TYPE sCmd :
STRUCT
	boStop : BOOL;
	boReset :BOOL;
	boJobReset: BOOL;
	boRFIDComplete: BOOL;
	boStartJob : BOOL;
	boTokenGrant :BOOL;
	boCancelCharging: BOOL;
END_STRUCT
END_TYPE

(* stored: Version 1.1.0.1, ProductVersion 3.1.4026.13
   DUT sCmd: Id {f4c04d97-f316-4286-bede-8829eadbf85e} *)
